(* IEC 61131-3 sources: plcassist-cli/packages/volt-lsp-iec/test-corpus/pro2193/Device/Plc Logic/Application/03 Hardware Units/31 SER/31.11 - Magazines/Main, 4 files *)

(* ---- Magazine_BeursFB.fb ---- *)
{attribute 'symbol' := 'none'}
FUNCTION_BLOCK Magazine_BeursFB
EXTENDS ModuleBaseHardwareFB
IMPLEMENTS IMagazineTransfer_Commands, IMagazineUnitSupply_Commands
VAR_INPUT
	xEmpty						: ARRAY[1..1] OF BOOL;
	{attribute 'symbol' := 'readwrite'}	Vacuum						: ARRAY[1..MaxVacuums] OF VacuumWithInputFB;
	{attribute 'symbol' := 'readwrite'}	BlowBetweenLabels			: ARRAY[1..MaxBlowBetweenLabels] OF ActuatorWithManualControlFB;
	motors						: IMagazineMotors_Commands;
	peeling						: IMagazinePeeling_Commands;
END_VAR
VAR_IN_OUT
	Data						: Magazine_Data;
END_VAR
VAR//VISU
END_VAR
VAR
	{attribute 'hide'}
	_anotherLabelNeeded			: BOOL;			// Private backing field for AnotherLabelNeeded property. Do not use directly.
END_VAR
VAR CONSTANT
	MaxVacuums					: USINT	:= 1;
	MaxBlowBetweenLabels		: USINT	:= 2;
	itfVacuums					: ARRAY[1..MaxVacuums] OF IVacuum :=[Vacuum[1]];
END_VAR

SUPER^();

END_FUNCTION_BLOCK

METHOD PROTECTED Alarms
VAR_INST
	SetError					: ARRAY[1..1] OF SetErrorFB;
END_VAR
SetError[1](
	moduleHandler	:= ModuleHandler,
	textRefId		:= MagazineBase_Errors,
	errorId			:= 1,		// Labelmagazine empty
	alarmCondition	:= PersistentVars.RecipeVars.EnableIML AND xEmpty[1],
	alarmDelay		:= 10.0,
	severity		:= enumErrorSeverity.Warning,
	reaction		:= enumErrorReaction.No_reaction,
	active			=> );
END_METHOD

METHOD PROTECTED Cyclic
VAR
	i	: USINT;
END_VAR
CycleTime[1](in := FALSE,	timeElapsed => rTimeActive,		timeMeasurement => );
CycleTime[2](in := FALSE,	timeElapsed => rTimeIdle,		timeMeasurement => );

FOR i := 1 TO MaxVacuums DO
	Vacuum[i](
		moduleHandler			:= ModuleHandler,
		manualControlEnabled	:= SER.ManualControlEnabled,
		textRefId				:= Vacuum_Label_Errors,
		errorId					:= i,
		alarmEnable				:= SER.DigIn.xAirPressureOK,
		alarmDelay				:= 3.0,
		severity				:= enumErrorSeverity.Fault,
		reaction				:= enumErrorReaction.No_reaction,
		refVacuumHighTime		:= ,
		refReleaseVacuumTime	:= Data.rPostReleaseLabelsDelay,
		input1					:= );
END_FOR

FOR i := 1 TO MaxBlowBetweenLabels DO
	BlowBetweenLabels[i](
		manualControlEnabled	:= SER.ManualControlEnabled);
END_FOR
END_METHOD

// Await a delay before releasing labels
METHOD PUBLIC DelayBeforeReleaseLabels : BOOL
VAR_INPUT
END_VAR
%FOLDER Commands/Transfer
IF ActState = enumMagazineState.None
OR ActState = enumMagazineState.ReadyWithLabels
OR ActState = enumMagazineState.ReadyWithoutLabels
THEN
	IF NOT xCommandDone THEN
		ActState := enumMagazineState.Transfer_DelayBeforeReleasingLabels;
	END_IF
END_IF

// Set command busy
xCommandBusy := TRUE;

// Return result when done
DelayBeforeReleaseLabels := xCommandDone;
END_METHOD

// Command to reset the module (Statemachine to zero state) in case of E-Stop
METHOD PUBLIC EStop : BOOL	// Returns true when drives are in standstill
%FOLDER Commands
ActState := enumMagazineState.None;

AnotherLabelNeeded := FALSE;

FOR i := 1 TO MaxBlowBetweenLabels DO
	BlowBetweenLabels[i].Reset();
END_FOR

Arrays.Vacuum_ReleaseAll(itfVacuums);

EStop := SUPER^.EStop();
END_METHOD

// After a state change, this method is called to execute the current state
METHOD PUBLIC Execute
CASE PersistentVars.RecipeVars.ActiveExchangeSet OF
	ExchangeSets.Default:
		Execute_Sequence1();
//	ExchangeSets.Product2, ExchangeSets.Product3:
//		Execute_Sequence2();
	ELSE
		ShowNoProgramWarning();
		Execute_Sequence1();
END_CASE
END_METHOD

METHOD PROTECTED Execute_Sequence1
VAR_INST
	Timer	: BTON;
END_VAR
IF xEntryActionActive THEN
	Timer.Reset();
END_IF

CASE ActState OF
	enumMagazineState.None:
		;
	enumMagazineState.ReadyWithLabels:
		;
	enumMagazineState.ReadyWithoutLabels:
		;

	enumMagazineState.Resetting_1:
		Resetting_1();
	enumMagazineState.Resetting_2:
		Resetting_2();

	enumMagazineState.GettingNewLabels:
		Arrays.Vacuum_ReleaseAll(itfVacuums);
		IF NOT peeling.LabelsPeeled THEN
			peeling.StartCommand();
		END_IF
		ActState := enumMagazineState.GetNew_MovingToTakeLabel;

	enumMagazineState.GetNew_MovingToTakeLabel:
		IF xEntryActionActive THEN
			motors.PrepareForImmediateNextCommand();
		END_IF

		IF motors.MoveToGetNewLabels(NOT peeling.LabelsPeeled) THEN
			ActState := enumMagazineState.GetNew_GettingAllLabels;
		END_IF

	enumMagazineState.GetNew_GettingAllLabels:
		peeling.ResetPeelingVacuums();
		IF GetAllLabels() THEN
			ActState := enumMagazineState.GetNew_MovingToWaitingPos;
		END_IF

	enumMagazineState.GetNew_MovingToWaitingPos:
		IF xEntryActionActive THEN
			motors.PrepareForImmediateNextCommand();
		END_IF

		// Start blowing when act drive position is NOT near position id 1 (rGetLabelsPos)
		FOR i := 1 TO MaxBlowBetweenLabels DO
			BlowBetweenLabels[i].SetOrReset(
				NOT motors.InPositionAt(
						position := MagazineMotors_Positions.getNewLabelsPos,
						tolerance := Data.rBlowBetweenLabelsDistance));
		END_FOR

		// Start peeling when leaving area
		IF NOT motors.InPositionAt(
			position	:= MagazineMotors_Positions.getNewLabelsPos,
			tolerance	:= 40)
		THEN
			peeling.StartCommand();
		END_IF

		IF motors.MoveToBeforeTakeoverLabels() THEN
			FOR i := 1 TO MaxBlowBetweenLabels DO
				BlowBetweenLabels[i].Reset();
			END_FOR
			xCommandDone := TRUE;
			IF HasPayload = enumPayload._All THEN
				ActState		:= enumMagazineState.ReadyWithLabels;
			ELSE
				ActState		:= enumMagazineState.ReadyWithoutLabels;
			END_IF
		END_IF

	enumMagazineState.Transfer_MovingToTakeover:
		IF motors.MoveToTakeoverLabels() THEN
			xCommandDone := TRUE;
			ActState := enumMagazineState.None;
		END_IF

	enumMagazineState.Transfer_DelayBeforeReleasingLabels:
		IF Timer.Set(TRUE, Data.rPreReleaseLabelsDelay) THEN
			xCommandDone := TRUE;
			ActState := enumMagazineState.None;
		END_IF

	enumMagazineState.Transfer_ReleasingLabels:
		ReleasingLabels();

END_CASE
END_METHOD

METHOD PROTECTED GetAllLabels : BOOL
%FOLDER States
FOR i := 1 TO MaxVacuums DO
	Vacuum[i].Set();
END_FOR

IF HasPayload = enumPayload._All THEN
	GetAllLabels := TRUE;
END_IF
END_METHOD

// Check if magazine needs to get new labels from the stockpile
METHOD PUBLIC GetNewLabels : BOOL
VAR_INPUT
END_VAR
%FOLDER Commands
// Ook met labels mag er een nieuw label gehaald worden. Bestaande labels worden afgeblazen.

IF (ActState = enumMagazineState.ReadyWithoutLabels OR ActState = enumMagazineState.ReadyWithLabels) AND NOT xCommandDone THEN
	ActState := enumMagazineState.GettingNewLabels;
END_IF

// Set command busy
xCommandBusy := TRUE;

// Return result when done
GetNewLabels := xCommandDone;
END_METHOD

// Move to a Takeover position. Parameter indicates number of Takeover position
METHOD PUBLIC MoveToTakeover : BOOL
VAR_INPUT
	iParameter : INT;	// 0: Invalid, 1: Takeover Pos 1, etc.
END_VAR
%FOLDER Commands/Transfer
IF ActState = enumMagazineState.None
OR ActState = enumMagazineState.ReadyWithLabels
OR ActState = enumMagazineState.ReadyWithoutLabels
THEN
	IF NOT xCommandDone THEN
		iCommandParameter := iParameter;	// Copy parameters

		ActState := enumMagazineState.Transfer_MovingToTakeover;
	END_IF
END_IF

// Set command busy
xCommandBusy := TRUE;

// Return result when done
MoveToTakeover := xCommandDone;
END_METHOD

{warning 'Add method implementation '}
METHOD MoveToWaitingPos : BOOL
%FOLDER Commands/Supply
END_METHOD

// Releases labels by resetting a vacuum. Parameter indicates which vacuums to kill
METHOD PUBLIC ReleaseLabels : BOOL
VAR_INPUT
	vacuumIndex		: WORD;	// 0: All vacuums, bit 1: Vacuum 1, bit 2: Vacuum 2, etc.
END_VAR
%FOLDER Commands/Supply
IF NOT CommandLock.Request(__POUNAME()) THEN
	RETURN;
END_IF

IF vacuumIndex = AllVacuums THEN	// Release all products by resetting all vacuums
	IF Arrays.Vacuum_ReleaseAll(itfVacuums) THEN
		ReleaseLabels	:= CommandLock.Release(__POUNAME());
	END_IF

ELSE						// Release a specific vacuum.
	IF Arrays.Vacuum_ReleaseSelected(itfVacuums, vacuumIndex) THEN
		ReleaseLabels	:= CommandLock.Release(__POUNAME());
	END_IF
END_IF
END_METHOD

METHOD PROTECTED ReleasingLabels
%FOLDER States
IF iCommandParameter = 0 THEN
	IF Arrays.Vacuum_ReleaseAll(itfVacuums) THEN
		xCommandDone := TRUE;
		ActState := enumMagazineState.None;
	END_IF

ELSE
	IF Arrays.Vacuum_ReleaseSelected(itfVacuums, iCommandParameter) THEN
		xCommandDone := TRUE;
		ActState := enumMagazineState.None;
	END_IF
END_IF
END_METHOD

// Command to reset the module. Servodrives are homed.
METHOD PUBLIC Reset : BOOL	// Returns true when homing done
%FOLDER Commands
IF ActState = enumMagazineState.None
OR ActState = enumMagazineState.ReadyWithLabels
OR ActState = enumMagazineState.ReadyWithoutLabels
THEN
	IF NOT xCommandDone THEN
		ActState := enumMagazineState.Resetting_1;		// Resetting		<-- Press F12 here
	END_IF
END_IF

// Set command busy
xCommandBusy := TRUE;

// Return result when done
Reset := xCommandDone;
END_METHOD

METHOD PROTECTED Resetting_1
%FOLDER States
IF xEntryActionActive THEN
	FOR i := 1 TO MaxBlowBetweenLabels DO
		BlowBetweenLabels[i].Reset();
	END_FOR

	Arrays.Vacuum_ResetIfNotHigh(itfVacuums);
END_IF

IF peeling.Reset() THEN
	ActState := enumMagazineState.Resetting_2;
END_IF
END_METHOD

METHOD PROTECTED Resetting_2
%FOLDER States
IF motors.Reset() THEN

	xCommandDone := TRUE;
	// Check if there are labels ready.
	ActState := SEL(	HasPayload = enumPayload._All,
						enumMagazineState.ReadyWithoutLabels,
						enumMagazineState.ReadyWithLabels);
END_IF
END_METHOD

METHOD PUBLIC SetDefaultData
%FOLDER Commands
Data.rPreReleaseLabelsDelay			:= 0.0;
Data.rPostReleaseLabelsDelay		:= 0.05;

Data.rBlowBetweenLabelsDistance		:= 10;

Data.rHammerOnTime					:= 0.2;
Data.rHammerOffTime					:= 0.5;
END_METHOD

// Start vacuums and transfer labels from the stockpile. Will time out in case of no vacuum detected
METHOD StartVacuums : enumResultGeneric
VAR_INPUT
	vacuumIndex		: WORD;	// 0: All vacuums, bit 1: Vacuum 1, bit 2: Vacuum 2, etc.
END_VAR
VAR_INST
	Timer			: BTON;
END_VAR
VAR
	i				: USINT;
END_VAR
%FOLDER Commands/Supply
IF NOT CommandLock.Request(__POUNAME()) THEN
	RETURN;
END_IF

IF CommandLock.FirstCall THEN
	Timer.Reset();
END_IF

IF Timer.Set(In := TRUE, Pt := 3) THEN	// Waiting for vacuum is taking too long
	StartVacuums		:= enumResultGeneric.Error;
	CommandLock.Release(__POUNAME());

ELSIF vacuumIndex = AllVacuums THEN	// Set all vacuums
	IF Arrays.Vacuum_SetAll(itfVacuums) THEN
		StartVacuums	:= enumResultGeneric.Success;
		CommandLock.Release(__POUNAME());
	END_IF

ELSE								// Set a specific vacuum.
	IF Arrays.Vacuum_SetSelected(itfVacuums, vacuumIndex) THEN
		StartVacuums	:= enumResultGeneric.Success;
		CommandLock.Release(__POUNAME());
	END_IF
END_IF
END_METHOD

// Command to reset the module (Statemachine to zero state)
METHOD PUBLIC Stop : BOOL	// Returns true when drives are in standstill
%FOLDER Commands
IF  ActState <> enumMagazineState.None
AND ActState <> enumMagazineState.ReadyWithLabels
AND ActState <> enumMagazineState.ReadyWithoutLabels
THEN
	ActState := enumMagazineState.None;
END_IF

AnotherLabelNeeded := FALSE;

FOR i := 1 TO MaxBlowBetweenLabels DO
	BlowBetweenLabels[i].Reset();
END_FOR
IF HasPayload <> enumPayload._All THEN
	Arrays.Vacuum_ReleaseAll(itfAdditionalVacuums);
END_IF

Arrays.Vacuum_ResetIfNotHigh(itfVacuums);

Stop := SUPER^.Stop();
END_METHOD

// Label transfer is complete. Reset the ReadyWithLabels state.
METHOD PUBLIC TransferComplete : BOOL
VAR_INPUT
	iParameter : INT := 0;	// Number indicates which transfer is completed
END_VAR
%FOLDER Commands
IF ActState = enumMagazineState.None AND NOT xCommandDone THEN

	// Move the motors back up to a safe position. This will be overwritten if IML is still enabled.
	motors.MoveToBeforeTakeoverLabels();

	// Signal the GetNewLabel process that another label is needed to complete the gripper.
	AnotherLabelNeeded := iParameter = 1;

	IF HasPayload = enumPayload.None THEN		// Reset Ready state only if all labels have been transferred.
		ActState := enumMagazineState.ReadyWithoutLabels;
	ELSE									// There is still 1 label on the magazine, so we are not yet ready to get new labels.
		ActState := enumMagazineState.ReadyWithLabels;
	END_IF

	TransferComplete := TRUE;
END_IF
END_METHOD

// When high, the magazine should get another label even if the cycle is in 'completing' mode. Another label is needed to complete the gripper.
{attribute 'monitoring':='call'}
PROPERTY AnotherLabelNeeded : BOOL
%FOLDER Properties
GET
VAR
END_VAR
AnotherLabelNeeded := _anotherLabelNeeded;
END_GET
SET
PRIVATE
VAR
END_VAR
_anotherLabelNeeded := AnotherLabelNeeded;
END_SET
END_PROPERTY

// Manual control of hardware is enabled from external context
{attribute 'monitoring':='call'}
PROPERTY ExternalManualControlEnabled : BOOL
%FOLDER Properties
SET
VAR
END_VAR
motors.ExternalManualControlEnabled		:= ExternalManualControlEnabled;
END_SET
END_PROPERTY

// The current payload status (products or labels) of the unit
{attribute 'monitoring':='call'}
PROPERTY HasPayload : enumPayload
%FOLDER Properties
GET
VAR
END_VAR
IF Arrays.Vacuum_All(
		vacuumArray	:= itfVacuums,
		condition	:= TRUE,
		channel		:= enumSelectIQ.Input)
THEN
	HasPayload := enumPayload._All;

ELSIF Arrays.Vacuum_Any(
		vacuumArray	:= itfVacuums,
		condition	:= TRUE,
		channel		:= enumSelectIQ.Both)
THEN
	HasPayload := enumPayload._Any;

ELSE
	HasPayload := enumPayload.None;
END_IF
END_GET
END_PROPERTY

(* ---- Magazine_DoubleM_WithFlipFB.fb ---- *)
// Drawer magazine with double M axes and Flip Label cylinder (for wrap labels)
{attribute 'symbol' := 'none'}
FUNCTION_BLOCK Magazine_DoubleM_WithFlipFB
EXTENDS Magazine_DoubleMFB
IMPLEMENTS IMagazine_Transfer_Commands, IMagazine_Supply_Commands
VAR_INPUT
	flipLabelSensorIn			: ARRAY[1..2] OF BOOL;
	flipLabelSensorOut			: ARRAY[1..2] OF BOOL;
	{attribute 'symbol' := 'readwrite'}	FlipLabel		: Cylinder_53ValveFB;
END_VAR

SUPER^(Data	:= Data);

END_FUNCTION_BLOCK

METHOD PROTECTED Cyclic
VAR
END_VAR
SUPER^.Cyclic();

FlipLabel(
	moduleHandler			:= ModuleHandler,
	manualControlEnabled	:= SER.ManualControlEnabled,
	textRefId				:= MagazineBase_Errors,
	errorId_SensorOut		:= 2,
	errorId_SensorIn		:= 3,
	alarmEnable				:= SER.DigIn.xAirPressureOK,
	alarmDelay				:= 10.0,
	severity				:= enumErrorSeverity.Fault,
	reaction				:= enumErrorReaction.No_reaction,
	inputOut				:= Arrays.Bool_All(flipLabelSensorOut, TRUE),
	inputIn					:= Arrays.Bool_All(flipLabelSensorIn, TRUE),
	rGiveAirToBothOutputs	:= 1.0,
	xEnableOutputs			:= TRUE);
END_METHOD

// Command to reset the module (ActStatemachine to zero state) in case of E-Stop
METHOD PUBLIC EStop : BOOL	// Returns true when drives are in standstill
%FOLDER Commands
FlipLabel.Reset();
EStop	:= SUPER^.EStop();
END_METHOD

// Gate open button is pushed. Safety gate is requesting to open (trigger signal)
METHOD PUBLIC GateOpenRequested
%FOLDER Commands/Gate Requests
FlipLabel.GoIn();
SUPER^.GateOpenRequested();
END_METHOD

// Check if magazine needs to get new labels from the stockpile
// A new label may also be obtained with labels already on the suction cups. Existing labels will be blown off.
METHOD PUBLIC GetNewLabels : BOOL
VAR_INPUT
	drawer	: enumDrawer;	// Choose which drawer (or other label stockpile) to get labels from
END_VAR
%FOLDER Commands/Magazine Supply
IF FlipLabel.GoIn() THEN
	GetNewLabels	:= SUPER^.GetNewLabels(drawer);
ELSE
	GetNewLabels	:= SUPER^.GetNewLabels(enumDrawer.NoDrawer);
END_IF
END_METHOD

// Move to a Waiting position.
METHOD PUBLIC MoveToSafeDistanceAboveDrawer : BOOL
%FOLDER Commands/Magazine
MoveToSafeDistanceAboveDrawer	:= FlipLabel.GoIn() AND_THEN SUPER^.MoveToSafeDistanceAboveDrawer();
END_METHOD

// Move to a Takeover position.
METHOD PUBLIC MoveToTakeOverPos : BOOL
VAR_INPUT
	takeOverPos	: USINT;	// 0: Invalid, 1: Takeover Pos 1, etc.
END_VAR
%FOLDER Commands/Magazine
// TEST! In case of lower drawer, the Flip can be set sooner.
IF  _activeDrawer = enumDrawer.Lower
AND Magazines.UnitMotors[1].actXPos > 200
AND Magazines.UnitMotors[1].actZPos < Magazines.DataMotors[1].getNewLabelsLowerPos.value - Magazines.DataMotors[1].SafeDistanceAboveDrawers - 100
THEN
	FlipLabel.GoOut();
END_IF

IF motors.InSafePos THEN
	FlipLabel.GoOut();
END_IF

IF NOT motors.InSafePos
AND NOT FlipLabel.IsIn
AND _activeDrawer <> enumDrawer.Lower
THEN
	LogPlc.Error('Movement unexpectedly halted because FlipLabel not in safe position');
	motors.Stop();
	RETURN;
END_IF

MoveToTakeOverPos	:= SUPER^.MoveToTakeOverPos(takeOverPos) AND_THEN FlipLabel.GoOut();
END_METHOD

// Move to waiting position.
METHOD PUBLIC MoveToWaitingPos : BOOL
%FOLDER Commands/Magazine
// TEST! In case of lower drawer, the Flip can be set sooner.
IF  _activeDrawer = enumDrawer.Lower
AND Magazines.UnitMotors[1].actXPos > 200
AND Magazines.UnitMotors[1].actZPos < Magazines.DataMotors[1].getNewLabelsLowerPos.value - Magazines.DataMotors[1].SafeDistanceAboveDrawers - 100
THEN
	FlipLabel.GoOut();
END_IF

IF motors.InSafePos THEN
	FlipLabel.GoOut();
END_IF

IF NOT motors.InSafePos
AND NOT FlipLabel.IsIn
AND _activeDrawer <> enumDrawer.Lower
THEN
	LogPlc.Error('Movement unexpectedly halted because FlipLabel not in safe position');
	motors.Stop();
	RETURN;
END_IF

MoveToWaitingPos	:= SUPER^.MoveToWaitingPos() AND_THEN FlipLabel.GoOut();
END_METHOD

// Command to reset the module. Servodrives are homed.
METHOD PUBLIC Reset : BOOL	// Returns true when homing done
%FOLDER Commands
Reset	:= FlipLabel.GoIn() AND_THEN SUPER^.Reset();
END_METHOD

// Command to reset the module (ActStatemachine to zero state)
METHOD PUBLIC Stop : BOOL	// Returns true when drives are in standstill
%FOLDER Commands
FlipLabel.GoIn();
Stop	:= SUPER^.Stop();
END_METHOD

// Label transfer is complete. Reset the ReadyWithLabels state.
METHOD PUBLIC TransferComplete : BOOL
VAR_INPUT
	iParameter : INT := 0;	// Number indicates which transfer is completed
END_VAR
%FOLDER Commands/Magazine Transfer
TransferComplete	:= FlipLabel.GoIn() AND_THEN SUPER^.TransferComplete();
END_METHOD

(* ---- Magazine_DoubleMFB.fb ---- *)
{attribute 'symbol' := 'none'}
FUNCTION_BLOCK Magazine_DoubleMFB
EXTENDS ModuleResettableFB
IMPLEMENTS IMagazine_Transfer_Commands, IMagazine_Supply_Commands, IModuleBlocksSafetyGate
VAR_INPUT
	{attribute 'symbol' := 'readwrite'}	Vacuum						: ARRAY[1..MaxVacuums] OF VacuumWithInputFB;
	{attribute 'symbol' := 'readwrite'}	VacuumAdditional			: ARRAY[1..MaxAdditionalVacuums] OF VacuumFB;
	{attribute 'symbol' := 'readwrite'}	BufferAir					: AirBufferFB;
	{attribute 'symbol' := 'readwrite'}	IonizingBar					: ActuatorWithManualControlFB;
	motors						: IMagazineMotors_Drawer_Commands;
END_VAR
VAR_IN_OUT
	Data						: Magazine_Data;
END_VAR
VAR//VISU
END_VAR
VAR
	{attribute 'hide'}
	_anotherLabelNeeded			: BOOL;			// Private backing field for property. Do not use directly.
	_activeDrawer				: enumDrawer;	// Private backing field for property. Do not use directly.
	_blowBetweenLabelsRequest	: BOOL;
	_activeState				: enumMagazineState;

	itfVacuums					: ARRAY[1..MaxVacuums] OF IVacuum;
	itfAdditionalVacuums		: ARRAY[1..MaxAdditionalVacuums] OF IVacuum;
	itfVacuumsTotal				: ARRAY[1..MaxVacuums + MaxAdditionalVacuums] OF IVacuum;
END_VAR
VAR CONSTANT
	MaxVacuums					: USINT	:= 6;
	MaxAdditionalVacuums		: USINT := 2;
END_VAR

SUPER^();

END_FUNCTION_BLOCK

METHOD PROTECTED Cyclic
VAR_INST
	testReset	: BOOL;
END_VAR
VAR
	i			: USINT;
END_VAR
FOR i := 1 TO MaxVacuums DO
	Vacuum[i](
		moduleHandler			:= ModuleHandler,
		manualControlEnabled	:= SER.ManualControlEnabled,
		textRefId				:= Vacuum_Label_Errors,
		errorId					:= i,
		alarmEnable				:= SER.DigIn.xAirPressureOK,
		alarmDelay				:= 3.0,
		severity				:= enumErrorSeverity.Fault,
		reaction				:= enumErrorReaction.No_reaction,
		refVacuumHighTime		:= ,
		refReleaseVacuumTime	:= Data.rPostReleaseLabelsDelay,
		input1					:= ,
		enableDuringSemiAuto	:= NOT SER.semiAutoInContinuousMode);
END_FOR

FOR i := 1 TO MaxAdditionalVacuums DO
	VacuumAdditional[i](
		moduleHandler			:= ModuleHandler,
		manualControlEnabled	:= SER.ManualControlEnabled,
		textRefId				:= Vacuum_Errors,
		alarmEnable				:= SER.DigIn.xAirPressureOK,
		alarmDelay				:= 3.0,
		severity				:= enumErrorSeverity.Fault,
		reaction				:= enumErrorReaction.No_reaction,
		refVacuumHighTime		:= ,
		refReleaseVacuumTime	:= Data.rPostReleaseLabelsDelay,
		enableDuringSemiAuto	:= NOT SER.semiAutoInContinuousMode);
END_FOR

BufferAir(
	manualControlEnabled	:= SER.ManualControlEnabled,
	vacuums					:= itfVacuumsTotal);

// Handle ionizing bar
IonizingBar(
	manualControlEnabled	:= FALSE);

IF SER.InAutomaticOperation_Rising THEN
	IonizingBar.Set();
END_IF

IF SER.InAutomaticOperation_Falling THEN
	IonizingBar.Reset();
END_IF

IF testReset AND_THEN Reset() THEN
	testReset	:= FALSE;
END_IF
END_METHOD

// Await a delay before releasing labels
METHOD PUBLIC DelayBeforeReleaseLabels : BOOL
VAR_INST
	Timer	: BTON;
END_VAR
%FOLDER Commands/Magazine Transfer
IF NOT CommandLock.Request(__POUNAME()) THEN
	RETURN;
END_IF

IF CommandLock.FirstCall THEN
	Timer.Reset();
END_IF

IF Timer.Set(TRUE, Data.rPreReleaseLabelsDelay) THEN
	DelayBeforeReleaseLabels	:= CommandLock.Release(__POUNAME());
END_IF
END_METHOD

// Command to reset the module (ActStatemachine to zero state) in case of E-Stop
METHOD PUBLIC EStop : BOOL	// Returns true when drives are in standstill
%FOLDER Commands
ActState := enumMagazineState.None;

AnotherLabelNeeded			:= FALSE;

Arrays.Vacuum_ReleaseAll(itfVacuums);
Arrays.Vacuum_ReleaseAll(itfAdditionalVacuums);

EStop := SUPER^.EStop();
END_METHOD

// Gate close button is released. Safety gate is cancelling request, so stop moving. (trigger signal)
METHOD PUBLIC GateCloseCancelled
%FOLDER Commands/Gate Requests
// Do nothing when gate closes
END_METHOD

// Gate close button is pushed. Safety gate is requesting to close (trigger signal)
METHOD PUBLIC GateCloseRequested
%FOLDER Commands/Gate Requests
// Do nothing when gate closes
END_METHOD

// Gate open button is released. Safety gate is cancelling request, so stop moving. (trigger signal)
METHOD PUBLIC GateOpenCancelled
%FOLDER Commands/Gate Requests
motors.Stop();
END_METHOD

// Gate open button is pushed. Safety gate is requesting to open (trigger signal)
METHOD PUBLIC GateOpenRequested
%FOLDER Commands/Gate Requests
motors.ProfileHomeToSafePosition();
motors.StartCommand();
END_METHOD

// Check if magazine needs to get new labels from the stockpile
// A new label may also be obtained with labels already on the suction cups. Existing labels will be blown off.
METHOD PUBLIC GetNewLabels : BOOL
VAR_INPUT
	drawer	: enumDrawer;	// Choose which drawer (or other label stockpile) to get labels from
END_VAR
VAR_INST
	localState			: SINT;
END_VAR
%FOLDER Commands/Magazine Supply
IF NOT CommandLock.Request(__POUNAME()) THEN
	RETURN;
END_IF

// Only update the local active drawer reference when a new drawer is known.... Not the best solution??..
IF drawer <> enumDrawer.LastDrawer THEN
	_activeDrawer		:= drawer;
END_IF

IF CommandLock.FirstCall THEN
	localState		:= 0;
	ActState		:= enumMagazineState.Busy_GetNew;
	motors.ProfileToHorizontal(_activeDrawer);
	ReleaseLabels(AllVacuums);
	ReleaseAdditionalVacuums(AllVacuums);
END_IF

CASE localState OF
	0:
		IF motors.StartCommand() THEN						// Movement done
			IF _activeDrawer = enumDrawer.NoDrawer THEN	// Wait for a drawer to be ready
				Increment.AnyInt(localState);
			ELSE
				GetNewLabels	:= CommandLock.Release(__POUNAME());
			END_IF
		END_IF
	1:
		IF _activeDrawer <> enumDrawer.NoDrawer THEN
			motors.ProfileToHorizontal(_activeDrawer);
			localState			:= 0;						// There is an active drawer, move again.
		END_IF
END_CASE
END_METHOD

METHOD PROTECTED Initialize
VAR
	i	: USINT;
	j	: USINT	:= 1;
END_VAR
SUPER^.Initialize();

// Set interfaces to correct vacuum instances
FOR i := 1 TO MaxAdditionalVacuums DO
	itfAdditionalVacuums[i]		:= VacuumAdditional[i];
END_FOR

FOR i := 1 TO MaxVacuums DO
	itfVacuums[i]				:= Vacuum[i];
	itfVacuumsTotal[i]			:= Vacuum[i];
END_FOR

IF MaxAdditionalVacuums > 0 THEN
	FOR i := MaxVacuums + 1 TO MaxVacuums + MaxAdditionalVacuums DO
		itfVacuumsTotal[i]		:= VacuumAdditional[j];
		Increment.AnyInt(j);
	END_FOR
END_IF
END_METHOD

// Move to a Waiting position.
METHOD PUBLIC MoveToSafeDistanceAboveDrawer : BOOL
%FOLDER Commands/Magazine
IF NOT CommandLock.Request(__POUNAME()) THEN
	RETURN;
END_IF

IF CommandLock.FirstCall THEN
	motors.ProfileSafeDistanceAboveDrawer(_activeDrawer);
END_IF

// Start blowing when act drive position is near position id 1 (rGetLabelsPos)
_blowBetweenLabelsRequest		:= motors.InPositionAt(
										position	:= MagazineMotors_Positions.getNewLabelsPos,
										tolerance	:= Data.rBlowBetweenLabelsDistance);

IF motors.StartCommand() THEN
	_blowBetweenLabelsRequest	:= FALSE;
	MoveToSafeDistanceAboveDrawer	:= CommandLock.Release(__POUNAME());
END_IF
END_METHOD

// Move to a Takeover position.
METHOD PUBLIC MoveToTakeOverPos : BOOL
VAR_INPUT
	takeOverPos	: USINT;	// 0: Invalid, 1: Takeover Pos 1, etc.
END_VAR
%FOLDER Commands/Magazine
IF takeOverPos < 1
OR takeOverPos > 4
THEN
	LogPlc.Error(CONCAT('Invalid parameter: ', TO_STRING(takeOverPos)));
	RETURN;
END_IF

IF NOT CommandLock.Request(__POUNAME()) THEN
	RETURN;
END_IF

IF CommandLock.FirstCall THEN
	// Check if already on correct Takeover position
	IF (takeOverPos = 1 AND_THEN motors.InPositionAt(position := MagazineMotors_Positions.takeover1Pos, tolerance := 1))
	OR (takeOverPos = 2 AND_THEN motors.InPositionAt(position := MagazineMotors_Positions.takeover2Pos, tolerance := 1))
	OR (takeOverPos = 3 AND_THEN motors.InPositionAt(position := MagazineMotors_Positions.takeover3Pos, tolerance := 1))
	OR (takeOverPos = 4 AND_THEN motors.InPositionAt(position := MagazineMotors_Positions.takeover4Pos, tolerance := 1))
	THEN
		IF HasPayload = enumPayload._All THEN
			ActState			:= enumMagazineState.ReadyWithLabels;
		ELSE
			ActState			:= enumMagazineState.ReadyWithoutLabels;
		END_IF
		MoveToTakeOverPos		:= CommandLock.Release(__POUNAME());
		RETURN;
	END_IF

	motors.ProfileToVertical(_activeDrawer, MagazineMotors_Positions.takeover1Pos);
END_IF

// Start blowing when act drive position is near position id 1 (rGetLabelsPos)
_blowBetweenLabelsRequest		:= motors.InPositionAt(
										position	:= MagazineMotors_Positions.getNewLabelsPos,
										tolerance	:= Data.rBlowBetweenLabelsDistance);

IF motors.StartCommand() THEN
	_blowBetweenLabelsRequest	:= FALSE;

	IF HasPayload = enumPayload._All THEN
		ActState				:= enumMagazineState.ReadyWithLabels;
	ELSE
		ActState				:= enumMagazineState.ReadyWithoutLabels;
	END_IF
	MoveToTakeOverPos			:= CommandLock.Release(__POUNAME());
END_IF
END_METHOD

// Move to waiting position.
METHOD PUBLIC MoveToWaitingPos : BOOL
%FOLDER Commands/Magazine
IF NOT CommandLock.Request(__POUNAME()) THEN
	RETURN;
END_IF

IF CommandLock.FirstCall THEN
	// Check if already on Waiting position
	IF motors.InPositionAt(position := MagazineMotors_Positions.waitingPosition, tolerance := 1) THEN
		IF HasPayload = enumPayload._All THEN
			ActState			:= enumMagazineState.ReadyWithLabels;
		ELSE
			ActState			:= enumMagazineState.ReadyWithoutLabels;
		END_IF
		MoveToWaitingPos		:= CommandLock.Release(__POUNAME());
		RETURN;
	END_IF

	motors.ProfileToVertical(_activeDrawer, MagazineMotors_Positions.waitingPosition);
END_IF

// Start blowing when act drive position is near position id 1 (rGetLabelsPos)
_blowBetweenLabelsRequest		:= motors.InPositionAt(
										position	:= MagazineMotors_Positions.getNewLabelsPos,
										tolerance	:= Data.rBlowBetweenLabelsDistance);

IF motors.StartCommand() THEN
	_blowBetweenLabelsRequest	:= FALSE;

	IF HasPayload = enumPayload._All THEN
		ActState				:= enumMagazineState.ReadyWithLabels;
	ELSE
		ActState				:= enumMagazineState.ReadyWithoutLabels;
	END_IF
	MoveToWaitingPos			:= CommandLock.Release(__POUNAME());
END_IF
END_METHOD

//
METHOD PUBLIC NewLabelsNeededDuringSemiAutoOperation
%FOLDER Commands/Magazine Transfer
ActState := enumMagazineState.LabelsNeededDuringSemiAuto;
END_METHOD

// Releases labels by resetting a vacuum. Parameter indicates which vacuums to kill
METHOD PUBLIC ReleaseAdditionalVacuums : BOOL
VAR_INPUT
	vacuumIndex		: WORD;	// 0: All vacuums, bit 1: Vacuum 1, bit 2: Vacuum 2, etc.
END_VAR
%FOLDER Commands/Magazine
IF vacuumIndex = AllVacuums THEN	// Release all products by resetting all vacuums
	IF Arrays.Vacuum_ReleaseAll(itfAdditionalVacuums) THEN
		ReleaseAdditionalVacuums	:= TRUE;
	END_IF

ELSE								// Release a specific vacuum.
	IF Arrays.Vacuum_ReleaseSelected(itfAdditionalVacuums, vacuumIndex) THEN
		ReleaseAdditionalVacuums	:= TRUE;
	END_IF
END_IF
END_METHOD

// Releases labels by resetting a vacuum. Parameter indicates which vacuums to kill
METHOD PUBLIC ReleaseLabels : BOOL
VAR_INPUT
	vacuumIndex		: WORD;	// 0: All vacuums, bit 1: Vacuum 1, bit 2: Vacuum 2, etc.
END_VAR
%FOLDER Commands/Magazine
IF vacuumIndex = AllVacuums THEN	// Release all products by resetting all vacuums
	IF Arrays.Vacuum_ReleaseAll(itfVacuums) THEN
		ReleaseLabels				:= TRUE;
	END_IF

ELSE								// Release a specific vacuum.
	IF Arrays.Vacuum_ReleaseSelected(itfVacuums, vacuumIndex) THEN
		ReleaseLabels				:= TRUE;
	END_IF
END_IF
END_METHOD

// Command to reset the module. Servodrives are homed.
METHOD PUBLIC Reset : BOOL	// Returns true when homing done
VAR_INST
	localState			: SINT;
	result				: UINT;
END_VAR
%FOLDER Commands
IF NOT CommandLock.Request(__POUNAME()) THEN
	RETURN;
END_IF

IF CommandLock.FirstCall THEN
	localState := 0;
	IF HasPayload <> enumPayload._All THEN
		Arrays.Vacuum_ReleaseAll(itfAdditionalVacuums);
	END_IF
	Arrays.Vacuum_ResetIfNotHigh(itfVacuums);
END_IF

CASE localState OF
	0:
		IF motors.Reset() THEN

			// Check if there are labels ready.
			IF HasPayload = enumPayload._All THEN
				ActState		:= enumMagazineState.ReadyWithLabels;
			ELSE
				ActState		:= enumMagazineState.ReadyWithoutLabels;
			END_IF

			Reset := CommandLock.Release(__POUNAME());
		END_IF
END_CASE
END_METHOD

// Releases labels by resetting a vacuum. Parameter indicates which vacuums to kill
METHOD PUBLIC StartAdditionalVacuums : BOOL
VAR_INPUT
	vacuumIndex		: WORD;	// 0: All vacuums, bit 1: Vacuum 1, bit 2: Vacuum 2, etc.
END_VAR
%FOLDER Commands/Magazine Supply
IF vacuumIndex = AllVacuums THEN	// Set all additional vacuums
	IF Arrays.Vacuum_SetAll(itfAdditionalVacuums) THEN
		StartAdditionalVacuums		:= TRUE;
	END_IF

ELSE								// Set a specific vacuum
	IF Arrays.Vacuum_SetSelected(itfAdditionalVacuums, vacuumIndex) THEN
		StartAdditionalVacuums		:= TRUE;
	END_IF
END_IF
END_METHOD

// Start vacuums and transfer labels from the stockpile. Will time out in case of no vacuum detected
METHOD StartVacuums : enumResultGeneric
VAR_INPUT
	vacuumIndex		: WORD;	// 0: All vacuums, bit 1: Vacuum 1, bit 2: Vacuum 2, etc.
END_VAR
VAR_INST
	Timer			: BTON;
END_VAR
VAR
	i				: USINT;
END_VAR
%FOLDER Commands/Magazine Supply
IF NOT CommandLock.Request(__POUNAME()) THEN
	RETURN;
END_IF

IF CommandLock.FirstCall THEN
	Timer.Reset();
END_IF

IF ser.semiAutoInContinuousMode THEN
	StartVacuums	:= enumResultGeneric.Success;
	CommandLock.Release(__POUNAME());
ELSIF Timer.Set(In := TRUE, Pt := 1) THEN	// Waiting for vacuum is taking too long
	StartVacuums		:= enumResultGeneric.Error;
	CommandLock.Release(__POUNAME());

ELSIF vacuumIndex = AllVacuums THEN	// Set all vacuums
	IF Arrays.Vacuum_SetAll(itfVacuums) THEN
		StartVacuums	:= enumResultGeneric.Success;
		CommandLock.Release(__POUNAME());
	END_IF

ELSE								// Set a specific vacuum.
	IF Arrays.Vacuum_SetSelected(itfVacuums, vacuumIndex) THEN
		StartVacuums	:= enumResultGeneric.Success;
		CommandLock.Release(__POUNAME());
	END_IF
END_IF
END_METHOD

// Command to reset the module (ActStatemachine to zero state)
METHOD PUBLIC Stop : BOOL	// Returns true when drives are in standstill
%FOLDER Commands
IF  ActState <> enumMagazineState.ReadyWithLabels
AND ActState <> enumMagazineState.ReadyWithoutLabels
THEN
	ActState := enumMagazineState.None;
END_IF

AnotherLabelNeeded := FALSE;

IF HasPayload <> enumPayload._All THEN
	Arrays.Vacuum_ReleaseAll(itfAdditionalVacuums);
END_IF
Arrays.Vacuum_ResetIfNotHigh(itfVacuums);

Stop := SUPER^.Stop();
END_METHOD

// Label transfer is complete. Reset the ReadyWithLabels state.
METHOD PUBLIC TransferComplete : BOOL
VAR_INPUT
	iParameter : INT := 0;	// Number indicates which transfer is completed
END_VAR
%FOLDER Commands/Magazine Transfer
// Signal the GetNewLabel process that another label is needed to complete the gripper.
AnotherLabelNeeded := iParameter = 1;

IF HasPayload = enumPayload.None THEN		// Reset Ready state only if all labels have been transferred.
	ActState := enumMagazineState.ReadyWithoutLabels;
ELSE										// There is still 1 label on the magazine, so we are not yet ready to get new labels.
	ActState := enumMagazineState.ReadyWithLabels;
END_IF

TransferComplete := TRUE;
END_METHOD

// Current state of magazine
{attribute 'monitoring':='call'}
PROPERTY ActState : enumMagazineState
%FOLDER Properties
GET
VAR
END_VAR
ActState := _activeState;
END_GET
SET
PROTECTED
VAR
END_VAR
_activeState := ActState;
END_SET
END_PROPERTY

// When high, the magazine should get another label even if the cycle is in 'completing' mode. Another label is needed to complete the gripper.
{attribute 'monitoring':='call'}
PROPERTY AnotherLabelNeeded : BOOL
%FOLDER Properties
GET
VAR
END_VAR
AnotherLabelNeeded := _anotherLabelNeeded;
END_GET
SET
PRIVATE
VAR
END_VAR
_anotherLabelNeeded := AnotherLabelNeeded;
END_SET
END_PROPERTY

// When high, the magazine should get another label even if the cycle is in 'completing' mode. Another label is needed to complete the gripper.
{attribute 'monitoring':='call'}
PROPERTY BlowBetweenLabelsRequest : BOOL
%FOLDER Properties
GET
VAR
END_VAR
BlowBetweenLabelsRequest := _blowBetweenLabelsRequest;
END_GET
END_PROPERTY

// Manual control of hardware is enabled from external context
{attribute 'monitoring':='call'}
PROPERTY ExternalManualControlEnabled : BOOL
%FOLDER Properties
SET
VAR
END_VAR
motors.ExternalManualControlEnabled		:= ExternalManualControlEnabled;
END_SET
END_PROPERTY

// The current payload status (products or labels) of the unit
{attribute 'monitoring':='call'}
PROPERTY HasPayload : enumPayload
%FOLDER Properties
GET
VAR
END_VAR
IF Arrays.Vacuum_All(
							vacuumArray	:= itfVacuums,
							condition	:= TRUE,
							channel		:= enumSelectIQ.Input)
//							channel		:= SEL(	SER.OperationMode = SER_OperationModeType.SemiAuto AND HMI.SemiAutoMode = enumSemiAutoModeType.WithoutVacuums,
//												enumSelectIQ.Input,
//												enumSelectIQ.Output))
THEN
	HasPayload := enumPayload._All;

ELSIF Arrays.Vacuum_Any(
							vacuumArray	:= itfVacuums,
							condition	:= TRUE,
							channel		:= enumSelectIQ.Both)
THEN
	HasPayload := enumPayload._Any;

ELSE
	HasPayload := enumPayload.None;
END_IF
END_GET
END_PROPERTY

// The axis is homed, and in a safe (parking) position
{attribute 'monitoring':='call'}
PROPERTY PUBLIC InSafePos : BOOL
%FOLDER Properties
GET
VAR
END_VAR
InSafePos := motors.InSafePos;
END_GET
END_PROPERTY

// Used by modules like: Z and M units, true when module is in a position where gate is free to open.
{attribute 'monitoring':='call'}
PROPERTY PUBLIC InSafePosForGate : BOOL
%FOLDER Commands/Gate Requests
GET
VAR
END_VAR
InSafePosForGate := motors.InPositionAt(MagazineMotors_Positions.middlePosition, 10);
END_GET
END_PROPERTY

(* ---- MagazineBaseFB.fb ---- *)
{attribute 'symbol' := 'none'}
FUNCTION_BLOCK MagazineBaseFB
EXTENDS ModuleBaseHardwareFB
IMPLEMENTS IMagazineTransfer_Commands, IMagazineUnitSupply_Commands
VAR_INPUT
	dwDisableCavityNumber		: DWORD;
	xEmpty						: ARRAY[1..2] OF BOOL;
	{attribute 'symbol' := 'readwrite'}	Vacuum						: ARRAY[1..MaxVacuums] OF VacuumWithPressureFB;
	{attribute 'symbol' := 'readwrite'}	Hammer						: ARRAY[1..MaxHammers] OF HammerFB;
	{attribute 'symbol' := 'readwrite'}	BufferAir					: AirBufferFB;
	{attribute 'symbol' := 'readwrite'}	BlowBetweenLabels			: ARRAY[1..MaxBlowBetweenLabels] OF ActuatorWithManualControlFB;
	motors						: IMagazineMotors_Commands;
END_VAR
VAR_IN_OUT
	Data						: Magazine_Data;
END_VAR
VAR//VISU
END_VAR
VAR
END_VAR
VAR CONSTANT
	MaxVacuums					: USINT	:= 4;
	MaxHammers					: USINT	:= MaxVacuums;
	MaxBlowBetweenLabels		: USINT	:= 1;
	itfVacuums					: ARRAY[1..MaxVacuums] OF IVacuum :=[Vacuum[1], Vacuum[2], Vacuum[3], Vacuum[4]];
	itfHammers					: ARRAY[1..MaxHammers] OF IActuator := [Hammer[1], Hammer[2], Hammer[3], Hammer[4]];
END_VAR

SUPER^();

END_FUNCTION_BLOCK

METHOD PROTECTED Alarms
END_METHOD

METHOD PROTECTED Cyclic
CycleTime[1](in := FALSE,	timeElapsed => rTimeActive,		timeMeasurement => );
CycleTime[2](in := FALSE,	timeElapsed => rTimeIdle,		timeMeasurement => );

FOR i := 1 TO MaxVacuums DO
	Vacuum[i](
		moduleHandler			:= ModuleHandler,
		manualControlEnabled	:= SER.ManualControlEnabled,
		textRefId				:= Vacuum_Errors,
		errorId					:= TO_WORD(i),
		alarmEnable				:= SER.DigIn.xAirPressureOK,
		alarmDelay				:= 3.0,
		severity				:= enumErrorSeverity.Fault,
		reaction				:= enumErrorReaction.No_reaction,
		refVacuumHighTime		:= ,
		refReleaseVacuumTime	:= Data.rPostReleaseLabelsDelay,
		input1					:= );
END_FOR

FOR i := 1 TO MaxHammers DO
	Hammer[i](
		moduleHandler			:= ModuleHandler,
		manualControlEnabled	:= SER.ManualControlEnabled,
		textRefId				:= MagazineBase_Errors,
		errorId					:= TO_UINT(i) + 10,
		alarmEnable				:= SER.DigIn.xAirPressureOK,
		alarmDelay				:= 0.0,
		severity				:= enumErrorSeverity.Fault,
		reaction				:= enumErrorReaction.No_reaction,
		rTimeLow				:= Data.rHammerOffTime,
		rTimeHigh				:= Data.rHammerOnTime,
		usiLimitStop			:= ,
		usiLimitAlarm			:= ,
		uiCounter				=> );
END_FOR

FOR i := 1 TO MaxBlowBetweenLabels DO
	BlowBetweenLabels[i](
		manualControlEnabled	:= SER.ManualControlEnabled);
END_FOR

BufferAir(
	manualControlEnabled		:= FALSE,
	vacuums						:= itfVacuums);
END_METHOD

// Await a delay before releasing labels
METHOD PUBLIC DelayBeforeReleaseLabels : BOOL
VAR_INPUT
END_VAR
%FOLDER Commands
IF ActState = enumMagazineState.None AND NOT xCommandDone THEN
	ActState := enumMagazineState.Transfer_DelayBeforeReleasingLabels;
END_IF

// Set command busy
xCommandBusy := TRUE;

// Return result when done
DelayBeforeReleaseLabels := xCommandDone;
END_METHOD

// Command to reset the module (Statemachine to zero state) in case of E-Stop
METHOD PUBLIC EStop : BOOL	// Returns true when drives are in standstill
%FOLDER Commands
ActState := enumMagazineState.None;

FOR i := 1 TO MaxBlowBetweenLabels DO
	BlowBetweenLabels[i].Reset();
END_FOR

Arrays.Vacuum_ReleaseAll(itfVacuums);

Arrays.Actuator_ResetAll(itfHammers);

EStop := SUPER^.EStop();
END_METHOD

// After a state change, this method is called to execute the current state
METHOD PUBLIC Execute
CASE PersistentVars.RecipeVars.ActiveExchangeSet OF
	ExchangeSets.Default:
		Execute_Sequence1();
//	ExchangeSets.Product2, ExchangeSets.Product3:
//		Execute_Sequence2();
	ELSE
		ShowNoProgramWarning();
		Execute_Sequence1();
END_CASE
END_METHOD

METHOD PROTECTED Execute_Sequence1
VAR_INST
	Timer	: BTON;
END_VAR
IF xEntryActionActive THEN
	Timer.Reset();
END_IF

CASE ActState OF
	enumMagazineState.None:
		;
	enumMagazineState.ReadyWithLabels:
		;
	enumMagazineState.ReadyWithoutLabels:
		;

	enumMagazineState.Resetting_1:
		Resetting_1();
	enumMagazineState.Resetting_2:
		Resetting_2();

	enumMagazineState.GettingNewLabels:
		Arrays.Vacuum_ReleaseAll(itfVacuums);
		ActState := enumMagazineState.GetNew_MovingToTakeLabel;

	enumMagazineState.GetNew_MovingToTakeLabel:
		IF motors.MoveToGetNewLabels() THEN
			ActState := enumMagazineState.GetNew_GettingAllLabels;
		END_IF

	enumMagazineState.GetNew_GettingAllLabels:
		IF GetAllLabels() THEN
			ActState := enumMagazineState.GetNew_MovingToWaitingPos;
		END_IF

	enumMagazineState.GetNew_MovingToWaitingPos:
		// Start blowing when act drive position is NOT near position id 1 (rGetLabelsPos)
		FOR i := 1 TO MaxBlowBetweenLabels DO
			BlowBetweenLabels[i].SetOrReset(
				NOT motors.InPositionAt(
						position := MagazineMotors_Positions.getNewLabelsPos,
						tolerance := Data.rBlowBetweenLabelsDistance));
		END_FOR

		IF motors.MoveToTakeoverLabels() THEN
			FOR i := 1 TO MaxBlowBetweenLabels DO
				BlowBetweenLabels[i].Reset();
			END_FOR
			xCommandDone := TRUE;
			ActState := SEL(HasPayload = enumPayload._All,
							enumMagazineState.ReadyWithoutLabels,
							enumMagazineState.ReadyWithLabels);
		END_IF

	enumMagazineState.Transfer_MovingToTakeover:
		IF motors.MoveToTakeoverLabels() THEN
			xCommandDone := TRUE;
			ActState := enumMagazineState.None;
		END_IF

	enumMagazineState.Transfer_DelayBeforeReleasingLabels:
		IF Timer.Set(TRUE, Data.rPreReleaseLabelsDelay) THEN
			xCommandDone := TRUE;
			ActState := enumMagazineState.None;
		END_IF

	enumMagazineState.Transfer_ReleasingLabels:
		ReleasingLabels();

END_CASE
END_METHOD

METHOD PROTECTED GetAllLabels : BOOL
VAR_INST
	Timer	: BTON;
END_VAR
%FOLDER States
IF xEntryActionActive THEN
	Timer.Reset();
END_IF

Timer.Set(TRUE, 0.3);
FOR i := 1 TO MaxVacuums DO
	IF Vacuum[i].HasPressure THEN
		Vacuum[i].Set();
		Hammer[i].Reset();
	ELSIF Timer.Q AND NOT Vacuum[i].IsTurnedOn THEN
		Hammer[i].Set();
	END_IF
END_FOR

IF HasPayload = enumPayload._All THEN
	GetAllLabels := TRUE;
END_IF
END_METHOD

// Check if magazine needs to get new labels from the stockpile
METHOD PUBLIC GetNewLabels : BOOL
VAR_INPUT
END_VAR
%FOLDER Commands
IF ActState = enumMagazineState.ReadyWithoutLabels AND NOT xCommandDone THEN
	ActState := enumMagazineState.GettingNewLabels;
END_IF

// Set command busy
xCommandBusy := TRUE;

// Return result when done
GetNewLabels := xCommandDone;
END_METHOD

// Move to a Takeover position. Parameter indicates number of Takeover position
METHOD PUBLIC MoveToTakeover : BOOL
VAR_INPUT
	iParameter : INT;	// 0: Invalid, 1: Takeover Pos 1, etc.
END_VAR
%FOLDER Commands
IF ActState = enumMagazineState.None
OR ActState = enumMagazineState.ReadyWithLabels
OR ActState = enumMagazineState.ReadyWithoutLabels
THEN
	IF NOT xCommandDone THEN
		iCommandParameter := iParameter;	// Copy parameters

		ActState := enumMagazineState.Transfer_MovingToTakeover;
	END_IF
END_IF

// Set command busy
xCommandBusy := TRUE;

// Return result when done
MoveToTakeover := xCommandDone;
END_METHOD

// Releases labels by resetting a vacuum. Parameter indicates which vacuums to kill
METHOD PUBLIC ReleaseLabels : BOOL
VAR_INPUT
	iParameter		: INT;	// 0: All vacuums, bit 1: Vacuum 1, bit 2: Vacuum 2, etc.
END_VAR
%FOLDER Commands
IF ActState = enumMagazineState.ReadyWithLabels AND NOT xCommandDone THEN
	iCommandParameter := iParameter;	// Copy parameters

	ActState := enumMagazineState.Transfer_ReleasingLabels;
END_IF

// Set command busy
xCommandBusy := TRUE;

// Return result when done
ReleaseLabels := xCommandDone;
END_METHOD

METHOD PROTECTED ReleasingLabels
%FOLDER States
IF iCommandParameter = 0 THEN
	IF Arrays.Vacuum_ReleaseAll(itfVacuums) THEN
		xCommandDone := TRUE;
		ActState := enumMagazineState.ReadyWithoutLabels;
	END_IF

ELSE
	IF Arrays.Vacuum_ReleaseSelected(itfVacuums, iCommandParameter) THEN

		xCommandDone := TRUE;

		IF Arrays.Vacuum_All(	vacuumArray	:= itfVacuums,
								condition	:= FALSE,
								channel		:= enumSelectIQ.Output)
		THEN	// Reset Ready state only if all labels have been transferred.
			ActState := enumMagazineState.ReadyWithoutLabels;
		ELSE	// There is still 1 label on the magazine, so we are not yet ready to get new labels.
			ActState := enumMagazineState.ReadyWithLabels;
		END_IF

	END_IF
END_IF
END_METHOD

// Command to reset the module. Servodrives are homed.
METHOD PUBLIC Reset : BOOL	// Returns true when homing done
%FOLDER Commands
IF ActState = enumMagazineState.None
OR ActState = enumMagazineState.ReadyWithLabels
OR ActState = enumMagazineState.ReadyWithoutLabels
THEN
	IF NOT xCommandDone THEN
		ActState := enumMagazineState.Resetting_1;		// Resetting		<-- Press F12 here
	END_IF
END_IF

// Set command busy
xCommandBusy := TRUE;

// Return result when done
Reset := xCommandDone;
END_METHOD

METHOD PROTECTED Resetting_1
%FOLDER States
IF xEntryActionActive THEN
	FOR i := 1 TO MaxBlowBetweenLabels DO
		BlowBetweenLabels[i].Reset();
	END_FOR

	Arrays.Vacuum_ReleaseAll(itfVacuums);

	Arrays.Actuator_ResetAll(itfHammers);
END_IF

ActState := enumMagazineState.Resetting_2;
END_METHOD

METHOD PROTECTED Resetting_2
%FOLDER States
IF motors.Reset() THEN
	xCommandDone := TRUE;
	ActState := enumMagazineState.ReadyWithoutLabels;
END_IF
END_METHOD

// Command to reset the module (Statemachine to zero state)
METHOD PUBLIC Stop : BOOL	// Returns true when drives are in standstill
%FOLDER Commands
IF  ActState <> enumMagazineState.None
AND ActState <> enumMagazineState.ReadyWithLabels
AND ActState <> enumMagazineState.ReadyWithoutLabels
THEN
	ActState := enumMagazineState.None;
END_IF

FOR i := 1 TO MaxBlowBetweenLabels DO
	BlowBetweenLabels[i].Reset();
END_FOR

Arrays.Actuator_ResetAll(itfHammers);
IF HasPayload <> enumPayload._All THEN
	Arrays.Vacuum_ReleaseAll(itfAdditionalVacuums);
END_IF
Arrays.Vacuum_ResetIfNotHigh(itfVacuums);

Stop := SUPER^.Stop();
END_METHOD

// Label transfer is complete. Reset the ReadyWithLabels state.
METHOD PUBLIC TransferComplete : BOOL
VAR_INPUT
	iParameter : INT := 0;	// Number indicates which transfer is completed
END_VAR
%FOLDER Commands
IF ActState = enumMagazineState.None AND NOT xCommandDone THEN

	IF HasPayload = enumPayload.None THEN		// Reset Ready state only if all labels have been transferred.
		ActState := enumMagazineState.ReadyWithoutLabels;
	ELSE									// There is still 1 label on the magazine, so we are not yet ready to get new labels.
		ActState := enumMagazineState.ReadyWithLabels;
	END_IF

	TransferComplete := TRUE;
END_IF
END_METHOD

// Manual control of hardware is enabled from external context
{attribute 'monitoring':='call'}
PROPERTY ExternalManualControlEnabled : BOOL
%FOLDER Properties
SET
VAR
END_VAR
motors.ExternalManualControlEnabled := ExternalManualControlEnabled;
END_SET
END_PROPERTY

// The current payload status (products or labels) of the unit
{attribute 'monitoring':='call'}
PROPERTY HasPayload : enumPayload
%FOLDER Properties
GET
VAR
END_VAR
IF Arrays.Vacuum_All(
		vacuumArray	:= itfVacuums,
		condition	:= TRUE,
		channel		:= enumSelectIQ.Input)
THEN
	HasPayload := enumPayload._All;

ELSIF Arrays.Vacuum_Any(
		vacuumArray	:= itfVacuums,
		condition	:= TRUE,
		channel		:= enumSelectIQ.Both)
THEN
	HasPayload := enumPayload._Any;

ELSE
	HasPayload := enumPayload.None;
END_IF
END_GET
END_PROPERTY
